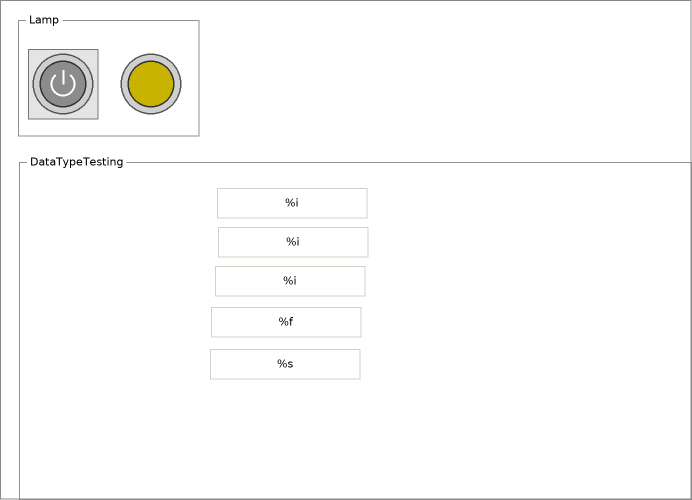
VISUALIZATION Visualization  // 692x500
    GroupBox (18,12 181x124), "Lamp"
        PowerSwitch (10,37 70x70), variable: MAIN.bStart, behaviour: TOGGLE, style: Switch-PowerSwitch-Gray
        Lamp1 (98,37 70x70), variable: MAIN.bEnable, style: Lamp-Lamp1-Yellow
    GroupBox (19,154 673x346), "DataTypeTesting"
        Textfield (198,34 150x30), "%i", text variable: MAIN.bEnable
        Textfield (199,73 150x30), "%i", text variable: MAIN.nINT
        Textfield (196,112 150x30), "%i", text variable: MAIN.nUINT
        Textfield (192,153 150x30), "%f", text variable: MAIN.fREAL
            OnMouseDown: write the text variable via Default
        Textfield (191,195 150x30), "%s", text variable: MAIN.sPowerStatus
            OnMouseDown: write the text variable via Default
END_VISUALIZATION

(* stored: Version 1.1.0.1, ProductVersion 3.1.4024.12
   Visu Visualization: Id {90c896e6-bbee-46bb-9860-014ab0e642ae} *)
